# B&R Automation Studio project DivertAlignmentTool (part 3)

#### WriteDivertTransform.st - not listed in the package file held
```iecst
(*********************************************************************************
 * Copyright: B&R Industrial Automation GmbH
 * Author:    nealj
 * Created:   November 30, 2023/4:29 PM
 *
 *********************************************************************************)

FUNCTION WriteDivertTransform
	// Clear the transform
	brsmemset(ADR(Schematic.Svg.Transform),0,SIZEOF(Schematic.Svg.Transform));
	// Add the opening bracket
	Schematic.Svg.Transform := '[';
	// Find the first filled divert entry and set its color
	FOR i:=0 TO NUM_DIVERTS DO
		IF Schematic.Diverts[i].Overlap <> 0 THEN
			RectName.Value := i;
			RectName.String := INT_TO_STRING(RectName.Value);
			brsmemset(ADR(NewLine),0,SIZEOF(NewLine));
			NewLine := '{"select":"#Div_';
			NewLine := CONCAT(NewLine,RectName.String);
			// If not found yet, set grey (0)
			IF NOT Schematic.Diverts[i].Found THEN
				NewLine := CONCAT(NewLine,'","fill":0,"duration":0}');
			// If found, but not measured, set blue (1)
			ELSIF Schematic.Diverts[i].Found AND NOT Schematic.Diverts[i].Measurements.Measured THEN
				NewLine := CONCAT(NewLine,'","fill":1,"duration":0}');
			// If found and measured, set blue (1)
			ELSIF Schematic.Diverts[i].Found AND Schematic.Diverts[i].Measurements.Measured THEN
				NewLine := CONCAT(NewLine,'","fill":2,"duration":0}');
			END_IF
			brsstrcat(ADR(Schematic.Svg.Transform),ADR(NewLine));
			EXIT;
		END_IF
	END_FOR
	// For all subsequent diverts, set the color
	FOR i:=(i+1) TO NUM_DIVERTS DO
		IF Schematic.Diverts[i].Overlap <> 0 THEN
			RectName.Value := i;
			RectName.String := INT_TO_STRING(RectName.Value);
			brsmemset(ADR(NewLine),0,SIZEOF(NewLine));
			NewLine := ',{"select":"#Div_';					// <-- Note the comma at the front of the string to separate it from the previous transform
			NewLine := CONCAT(NewLine,RectName.String);
			// If not found yet, set grey (0)
			IF NOT Schematic.Diverts[i].Found THEN
				NewLine := CONCAT(NewLine,'","fill":0,"duration":0}');
				// If found, but not measured, set blue (1)
			ELSIF Schematic.Diverts[i].Found AND NOT Schematic.Diverts[i].Measurements.Measured THEN
				NewLine := CONCAT(NewLine,'","fill":1,"duration":0}');
				// If found and measured, set blue (1)
			ELSIF Schematic.Diverts[i].Found AND Schematic.Diverts[i].Measurements.Measured THEN
				NewLine := CONCAT(NewLine,'","fill":2,"duration":0}');
			END_IF
			brsstrcat(ADR(Schematic.Svg.Transform),ADR(NewLine));
		END_IF
	END_FOR
	// Add the closing bracket
	NewLine := ']';
	brsstrcat(ADR(Schematic.Svg.Transform),ADR(NewLine));

END_FUNCTION
```

### SampleTrakCode.var - Variables for the example trak program
```iecst
(*
Array of all segment references*)
VAR
	SegmentRefs : ARRAY[0..NUM_SEGMENTS] OF UDINT;
END_VAR
(*
Motion Parameters*)
VAR
	MotionParameters : ShMotionParType;
END_VAR
```

### Program Logical/SampleTrakCode/AssemblyCtrl (IEC) - The main task for the example trak program

#### Cyclic.st - Cyclic code
```iecst
PROGRAM _CYCLIC

	CASE AsmState OF

		// When the controller starts up, power on the trak
		ASM_IDLE:
			AsmReadInfo.Enable := TRUE;
			AsmReadStatus.Enable := TRUE;
			AsmState := ASM_POWER_ON;

		// If needed, power on the assembly and wait for it to power on
		ASM_POWER_ON:
			IF NOT AsmReadInfo.AssemblyInfo.PowerOn THEN
				AsmPowerOn.Execute := TRUE;
			ELSIF AsmReadInfo.AssemblyInfo.PowerOn AND AsmReadStatus.AssemblyReady THEN
				AsmPowerOn.Execute := FALSE;
				AsmState := ASM_FIND_ALL_SHUTTLES;
			END_IF

		// Wait for the start command, then get a list of all shuttles on the trak. Skip to ASM_RUNNING if there are no shuttles
		ASM_FIND_ALL_SHUTTLES:
			IF gStartTrak THEN
				AsmGetShuttle.Enable := TRUE;
				IF AsmGetShuttle.Valid THEN
					IF AsmGetShuttle.TotalCount > 0 THEN
						AsmState := ASM_READ_FROM_SHUTTLE;
					ELSE
						AsmGetShuttle.Enable := FALSE;
						AsmState := ASM_RUNNING;
					END_IF
				END_IF
			END_IF

		ASM_READ_FROM_SHUTTLE:
			AsmGetShuttle.Next := FALSE;
			// Read the userdata from the shuttle
			ShCopyUserData.Axis := ADR(AsmGetShuttle.Axis);
			ShCopyUserData.DataAddress := ADR(UserData);
			ShCopyUserData.DataSize := SIZEOF(UserData);
			ShCopyUserData.Mode := mcACPTRAK_USERDATA_GET;
			ShCopyUserData.Execute := TRUE;
			IF ShCopyUserData.Done THEN
				ShCopyUserData.Execute := FALSE;
				AsmState := ASM_WRITE_TO_SHUTTLE;
			END_IF

		// Make the shuttle grey, set its destination, and assign it a serial number
		ASM_WRITE_TO_SHUTTLE:
			// Set up intital userdata
			UserData.Red := 0.5;
			UserData.Green := 0.5;
			UserData.Blue := 0.5;
			IF UserData.ShuttleSerialNum = '' THEN
				SN_String := '';
				SN_Index := SN_Index + 1;
				SN_IndexStr := USINT_TO_STRING(SN_Index);
				SN_String := CONCAT(SN_String,SN_Prefix);
				SN_String := CONCAT(SN_String,SN_IndexStr);
				UserData.ShuttleSerialNum := SN_String;
			END_IF
			// Write the userdata to the shuttle
			ShCopyUserData.Axis := ADR(AsmGetShuttle.Axis);
			ShCopyUserData.DataAddress := ADR(UserData);
			ShCopyUserData.DataSize := SIZEOF(UserData);
			ShCopyUserData.Mode := mcACPTRAK_USERDATA_SET;
			ShCopyUserData.Execute := TRUE;
			IF ShCopyUserData.Done THEN
				ShCopyUserData.Execute := FALSE;
				AsmState := ASM_MOVE_SHUTTLE;
			END_IF

		// Send the shuttle to the destination defined above
		ASM_MOVE_SHUTTLE:
			RoutedMoveAbs.Axis := ADR(AsmGetShuttle.Axis);
			RoutedMoveAbs.Sector := ADR(SEC_MainLoop);
			RoutedMoveAbs.Position := 0.00;
			RoutedMoveAbs.Velocity := MotionParameters.Velocity;
			RoutedMoveAbs.Acceleration := MotionParameters.Acceleration;
			RoutedMoveAbs.Deceleration := MotionParameters.Deceleration;
			RoutedMoveAbs.AdvancedParameters.StartDirection := mcDIR_POSITIVE;
			RoutedMoveAbs.AdvancedParameters.EndDirection := mcDIR_POSITIVE;
			RoutedMoveAbs.AdvancedParameters.NumberOfTransitPoints := 0;
			RoutedMoveAbs.Execute := TRUE;
			AsmState := ASM_CHECK_FOR_MORE;

		// Once the move is active, check for remaining shuttles
		ASM_CHECK_FOR_MORE:
			IF RoutedMoveAbs.Active THEN
				RoutedMoveAbs.Execute := FALSE;
				IF AsmGetShuttle.RemainingCount > 0 THEN
					AsmGetShuttle.Next := TRUE;
					AsmState := ASM_READ_FROM_SHUTTLE;
				ELSE
					AsmGetShuttle.Enable := FALSE;
					AsmState := ASM_RUNNING;
				END_IF
			END_IF

		// All shuttles have been put in motion
		ASM_RUNNING:
			// Reset the start command
			gStartTrak := FALSE;
			// If the stop command is issued, stop all shuttles
			IF gStopTrak THEN
				AsmStop.Execute := TRUE;
				IF AsmStop.Done THEN
					AsmStop.Execute := FALSE;
					AsmState := ASMSTOP_FIND_ALL_SHUTTLES;
				END_IF
			END_IF

		// ===========================================================
		// GET ALL SHUTTLES TO BE STOPPED AT THE START OF THE TOP LOOP
		// ===========================================================
		// Get a list of all shuttles on the trak. Skip to ASM_RUNNING if there are no shuttles
		ASMSTOP_FIND_ALL_SHUTTLES:
			AsmGetShuttle.Enable := TRUE;
			IF AsmGetShuttle.Valid THEN
				IF AsmGetShuttle.TotalCount > 0 THEN
					AsmState := ASMSTOP_READ_FROM_SHUTTLE;
				ELSE
					AsmGetShuttle.Enable := FALSE;
					gStopTrak := FALSE;
					AsmState := ASM_IDLE;
				END_IF
			END_IF

		ASMSTOP_READ_FROM_SHUTTLE:
			AsmGetShuttle.Next := FALSE;
			// Read the userdata from the shuttle
			ShCopyUserData.Axis := ADR(AsmGetShuttle.Axis);
			ShCopyUserData.DataAddress := ADR(UserData);
			ShCopyUserData.DataSize := SIZEOF(UserData);
			ShCopyUserData.Mode := mcACPTRAK_USERDATA_GET;
			ShCopyUserData.Execute := TRUE;
			IF ShCopyUserData.Done THEN
				ShCopyUserData.Execute := FALSE;
				AsmState := ASMSTOP_WRITE_TO_SHUTTLE;
			END_IF

		// Make the shuttle black, and set its destination
		ASMSTOP_WRITE_TO_SHUTTLE:
			// Set userdata to reflect the stop
			UserData.Red := 0.0;
			UserData.Green := 0.0;
			UserData.Blue := 0.0;
			// Write the userdata to the shuttle
			ShCopyUserData.Axis := ADR(AsmGetShuttle.Axis);
			ShCopyUserData.DataAddress := ADR(UserData);
			ShCopyUserData.DataSize := SIZEOF(UserData);
			ShCopyUserData.Mode := mcACPTRAK_USERDATA_SET;
			ShCopyUserData.Execute := TRUE;
			IF ShCopyUserData.Done THEN
				ShCopyUserData.Execute := FALSE;
				AsmState := ASMSTOP_MOVE_SHUTTLE;
			END_IF

		// Send the shuttle to the destination defined above
		ASMSTOP_MOVE_SHUTTLE:
			RoutedMoveAbs.Axis := ADR(AsmGetShuttle.Axis);
			RoutedMoveAbs.Sector := ADR(SEC_MainLoop);
			RoutedMoveAbs.Position := 0.00;
			RoutedMoveAbs.Velocity := MotionParameters.Velocity;
			RoutedMoveAbs.Acceleration := MotionParameters.Acceleration;
			RoutedMoveAbs.Deceleration := MotionParameters.Deceleration;
			RoutedMoveAbs.AdvancedParameters.StartDirection := mcDIR_UNDEFINED;
			RoutedMoveAbs.AdvancedParameters.EndDirection := mcDIR_POSITIVE;
			RoutedMoveAbs.Execute := TRUE;
			AsmState := ASMSTOP_CHECK_FOR_MORE;

		// Once the move is active, check for remaining shuttles
		ASMSTOP_CHECK_FOR_MORE:
			IF RoutedMoveAbs.Active THEN
				RoutedMoveAbs.Execute := FALSE;
				IF AsmGetShuttle.RemainingCount > 0 THEN
					AsmGetShuttle.Next := TRUE;
					AsmState := ASMSTOP_READ_FROM_SHUTTLE;
				ELSE
					AsmGetShuttle.Enable := FALSE;
					gStopTrak := FALSE;
					AsmState := ASM_IDLE;
				END_IF
			END_IF

		// Example error state
		ASM_ERROR:

	END_CASE

	// Call FUBs
	AsmPowerOn();
	AsmPowerOff();
	AsmReadInfo();
	AsmReadStatus();
	AsmGetShuttle();
	AsmStop();
	ShCopyUserData();
	RoutedMoveAbs();
	SecAddShuttle();

END_PROGRAM
```

#### Init.st - Init code
```iecst
PROGRAM _INIT

	// Set up assembly FUBs
	AsmPowerOn.Assembly := ADR(gAssembly_1);
	AsmPowerOff.Assembly := ADR(gAssembly_1);
	AsmReadInfo.Assembly := ADR(gAssembly_1);
	AsmReadStatus.Assembly := ADR(gAssembly_1);
	AsmGetShuttle.Assembly := ADR(gAssembly_1);
	AsmStop.Assembly := ADR(gAssembly_1);
	AsmStop.StopMode := mcSTOPMODE_JERK_LIMIT;

	//Set up shuttle spawning FUB
	SecAddShuttle.Sector := ADR(SEC_MainLoop);
	SecAddShuttle.Position := 0.00;

	// Set motion parameters
	MotionParameters.Velocity     := 1.0;
	MotionParameters.Acceleration := 40.0;
	MotionParameters.Deceleration := 40.0;

	// List all segment references
	SegmentRefs[1] := ADR(SEG_001);
	SegmentRefs[2] := ADR(SEG_002);
	SegmentRefs[3] := ADR(SEG_003);
	SegmentRefs[4] := ADR(SEG_004);
	SegmentRefs[5] := ADR(SEG_005);
	SegmentRefs[6] := ADR(SEG_006);
	SegmentRefs[7] := ADR(SEG_007);
	SegmentRefs[8] := ADR(SEG_008);
	SegmentRefs[9] := ADR(SEG_009);
	SegmentRefs[10] := ADR(SEG_010);
	SegmentRefs[11] := ADR(SEG_011);
	SegmentRefs[12] := ADR(SEG_012);
	SegmentRefs[13] := ADR(SEG_013);
	SegmentRefs[14] := ADR(SEG_014);
	SegmentRefs[15] := ADR(SEG_015);
	SegmentRefs[16] := ADR(SEG_016);
	SegmentRefs[17] := ADR(SEG_017);
	SegmentRefs[18] := ADR(SEG_018);
	SegmentRefs[19] := ADR(SEG_019);
	SegmentRefs[20] := ADR(SEG_020);
	SegmentRefs[21] := ADR(SEG_021);
	SegmentRefs[22] := ADR(SEG_022);
	SegmentRefs[23] := ADR(SEG_023);
	SegmentRefs[24] := ADR(SEG_024);
	SegmentRefs[25] := ADR(SEG_025);
	SegmentRefs[26] := ADR(SEG_026);
	SegmentRefs[27] := ADR(SEG_027);
	SegmentRefs[28] := ADR(SEG_028);
	SegmentRefs[29] := ADR(SEG_029);
	SegmentRefs[30] := ADR(SEG_030);
	SegmentRefs[31] := ADR(SEG_031);
	SegmentRefs[32] := ADR(SEG_032);
	SegmentRefs[33] := ADR(SEG_033);
	SegmentRefs[34] := ADR(SEG_034);
	SegmentRefs[35] := ADR(SEG_035);
	SegmentRefs[36] := ADR(SEG_036);
	SegmentRefs[37] := ADR(SEG_037);
	SegmentRefs[38] := ADR(SEG_038);
	SegmentRefs[39] := ADR(SEG_039);
	SegmentRefs[40] := ADR(SEG_040);
	SegmentRefs[41] := ADR(SEG_041);
	SegmentRefs[42] := ADR(SEG_042);
	SegmentRefs[43] := ADR(SEG_043);
	SegmentRefs[44] := ADR(SEG_044);
	SegmentRefs[45] := ADR(SEG_045);
	SegmentRefs[46] := ADR(SEG_046);
	SegmentRefs[47] := ADR(SEG_047);
	SegmentRefs[48] := ADR(SEG_048);
	SegmentRefs[49] := ADR(SEG_049);
	SegmentRefs[50] := ADR(SEG_050);
	SegmentRefs[51] := ADR(SEG_051);
	SegmentRefs[52] := ADR(SEG_052);
	SegmentRefs[53] := ADR(SEG_053);
	SegmentRefs[54] := ADR(SEG_054);
	SegmentRefs[55] := ADR(SEG_055);
	SegmentRefs[56] := ADR(SEG_056);
	SegmentRefs[57] := ADR(SEG_057);
	SegmentRefs[58] := ADR(SEG_058);
	SegmentRefs[59] := ADR(SEG_059);
	SegmentRefs[60] := ADR(SEG_060);
	SegmentRefs[61] := ADR(SEG_061);
	SegmentRefs[62] := ADR(SEG_062);
	SegmentRefs[63] := ADR(SEG_063);
	SegmentRefs[64] := ADR(SEG_064);
	SegmentRefs[65] := ADR(SEG_065);
	SegmentRefs[66] := ADR(SEG_066);
	SegmentRefs[67] := ADR(SEG_067);
	SegmentRefs[68] := ADR(SEG_068);
	SegmentRefs[69] := ADR(SEG_069);
	SegmentRefs[70] := ADR(SEG_070);
	SegmentRefs[71] := ADR(SEG_071);
	SegmentRefs[72] := ADR(SEG_072);
	SegmentRefs[73] := ADR(SEG_073);
	SegmentRefs[74] := ADR(SEG_074);
	SegmentRefs[75] := ADR(SEG_075);
	SegmentRefs[76] := ADR(SEG_076);
	SegmentRefs[77] := ADR(SEG_077);
	SegmentRefs[78] := ADR(SEG_078);
	SegmentRefs[79] := ADR(SEG_079);
	SegmentRefs[80] := ADR(SEG_080);
	SegmentRefs[81] := ADR(SEG_081);
	SegmentRefs[82] := ADR(SEG_082);
	SegmentRefs[83] := ADR(SEG_083);

	// List of all sectors (to avoid warnings in the logger)
	SEC_MainLoop;
	SEC_RedHerring_1;
	SEC_SecondLoop;
	SEC_VolcanoLeft;
	SEC_VolcanoRight;
	SEC_Squiggle;
	SEC_FlipFlop;
	SEC_RedHerring_2;
	SEC_MaintenanceLoop;

END_PROGRAM
```

#### Types.typ - Local data types
```iecst
TYPE
	AsmStateEnum :
		( (*State of the assembly control task*)
		ASM_IDLE,
		ASM_POWER_ON,
		ASM_FIND_ALL_SHUTTLES,
		ASM_READ_FROM_SHUTTLE,
		ASM_TRACK_SHUTTLE,
		ASM_WRITE_TO_SHUTTLE,
		ASM_MOVE_SHUTTLE,
		ASM_CHECK_FOR_MORE,
		ASM_RUNNING,
		ASMSTOP_FIND_ALL_SHUTTLES,
		ASMSTOP_READ_FROM_SHUTTLE,
		ASMSTOP_WRITE_TO_SHUTTLE,
		ASMSTOP_MOVE_SHUTTLE,
		ASMSTOP_CHECK_FOR_MORE,
		ASM_ERROR
		);
END_TYPE
```

#### Variables.var - Local variables
```iecst
(*Assembly variables*)
VAR
	AsmPowerOn : MC_BR_AsmPowerOn_AcpTrak; (*FUB to power on the assembly*)
	AsmPowerOff : MC_BR_AsmPowerOff_AcpTrak; (*FUB to power off the assembly*)
	AsmReadInfo : MC_BR_AsmReadInfo_AcpTrak; (*FUB to read the information of the assembly*)
	AsmReadStatus : MC_BR_AsmReadStatus_AcpTrak; (*FUB to read the status of the assembly*)
	AsmGetShuttle : MC_BR_AsmGetShuttle_AcpTrak; (*FUB to get references for all shuttles on the assembly*)
	AsmStop : MC_BR_AsmStop_AcpTrak; (*FUB to get references for all shuttles on the assembly*)
	AsmState : AsmStateEnum; (*State of the assembly control task*)
	SecAddShuttle : MC_BR_SecAddShuttle_AcpTrak;
END_VAR
(*
Shuttle variables*)
VAR
	ShCopyUserData : MC_BR_ShCopyUserData_AcpTrak; (*FUB for the initial writing of data during startup*)
	UserData : UserDataType; (*Structure for the initial writing of data during startup*)
	RoutedMoveAbs : MC_BR_RoutedMoveAbs_AcpTrak; (*FUB to move the shuttles on the trak to their first station*)
END_VAR
(*
Variables for serial number generation*)
VAR
	SN_Prefix : STRING[9] := 'TEST_SN_'; (*The prefix for all generated serial numbers*)
	SN_Index : USINT := 0; (*The number to be assigned to each shuttle (as a number)*)
	SN_IndexStr : STRING[4]; (*The number to be assigned to each shuttle (as a string)*)
	SN_String : STRING[12]; (*The string of the serial number to be assigned to each shuttle*)
END_VAR
```

#### Exit.st
```iecst
PROGRAM _EXIT

	RoutedMoveAbs.Execute := FALSE;
	RoutedMoveAbs();

END_PROGRAM
```

### Program Logical/DivertAlignment/GatherInfo (IEC)

#### Types.typ
```iecst
TYPE
	GatherStateEnum :
		(
		GATHER_IDLE,
		GATHER_SEG_AND_SEC,
		GATHER_SEG_AND_SEC_INFO,
		GATHER_DIVERTS,
		GATHER_SHUTTLE,
		GATHER_MOVE_TO_START,
		GATHER_MOVE_ALONG_SEC,
		GATHER_MONITOR_FOR_MIDPOINT,
		GATHER_ACKNOWLEDGE,
		GATHER_DONE
		);
END_TYPE
```

#### Variables.var
```iecst
VAR
	GatherState : GatherStateEnum;
	AssemblySchematics : AsmSchemType;
END_VAR
(*
FUBs and Vars for getting segments and their information*)
VAR
	AsmGetSeg : MC_BR_AsmGetSegment_AcpTrak;
	SecStop : MC_BR_SecStop_AcpTrak;
	SegGetInfo : MC_BR_SegGetInfo_AcpTrak;
	SecGetInfo : MC_BR_SecGetInfo_AcpTrak;
	CmdGather : BOOL;
	CmdContinue : BOOL;
	AsmGetSec : MC_BR_AsmGetSector_AcpTrak;
END_VAR
(*
FUBs and Vars for moving the shuttle around the trak*)
VAR
	AsmGetShuttle : MC_BR_AsmGetShuttle_AcpTrak;
	RoutedMoveAbs : MC_BR_RoutedMoveAbs_AcpTrak;
	ElasticMoveAbs : MC_BR_ElasticMoveAbs_AcpTrak;
	ShReadInfo : MC_BR_ShReadInfo_AcpTrak;
	ShReadSeg : MC_BR_ShReadSegmentInfo_AcpTrak;
	TestVelocity : REAL := 1.0;
	DivertIndex : UINT;
	SectorIndex : UINT;
	AcknowledgeTimer : TON;
	AcknowledgeTime : TIME := T#400ms;
END_VAR
```

#### Cyclic.st
```iecst
PROGRAM _CYCLIC
	(* Insert code here *)
	CASE GatherState OF
		GATHER_IDLE:
			// Wait for command, then clear the schematic structure and enable the AsmGetSeg and AsmGetSec FUBs
			IF CmdGather THEN
				brsmemset(ADR(AssemblySchematics),0,SIZEOF(AssemblySchematics));
				AsmGetSeg.Enable := TRUE;
				AsmGetSec.Enable := TRUE;
				GatherState := GATHER_SEG_AND_SEC;
			END_IF

		GATHER_SEG_AND_SEC:
			// Wait for validity
			IF AsmGetSeg.Valid AND AsmGetSec.Valid THEN
				// Clear the "next" signals
				AsmGetSeg.Next := FALSE;
				AsmGetSec.Next := FALSE;
				// Plug the segment and sectors into the respective get infor FUBs
				SegGetInfo.Segment := ADR(AsmGetSeg.Segment);
				SecGetInfo.Sector := ADR(AsmGetSec.Sector);
				// Execute the FUBs
				SegGetInfo.Execute := TRUE;
				SecGetInfo.Execute := TRUE;
				GatherState := GATHER_SEG_AND_SEC_INFO;
			END_IF

		GATHER_SEG_AND_SEC_INFO:
			// Wait for the SegGetInfo and SecGetInfo FUBs to finish
			IF SegGetInfo.Done AND SecGetInfo.Done THEN
				// Record the segment information (use the segment ID as the index)
				AssemblySchematics.Segment[SegGetInfo.SegmentInfo.ID].Reference := AsmGetSeg.Segment;
				AssemblySchematics.Segment[SegGetInfo.SegmentInfo.ID].Name := SegGetInfo.SegmentInfo.Name;
				AssemblySchematics.Segment[SegGetInfo.SegmentInfo.ID].ID := SegGetInfo.SegmentInfo.ID;
				AssemblySchematics.Segment[SegGetInfo.SegmentInfo.ID].Type := SegGetInfo.SegmentInfo.Type;
				AssemblySchematics.Segment[SegGetInfo.SegmentInfo.ID].StartFrame := SegGetInfo.SegmentInfo.StartFrame;
				AssemblySchematics.Segment[SegGetInfo.SegmentInfo.ID].EndFrame := SegGetInfo.SegmentInfo.EndFrame;
				// Record the sector information (store them in the order they are found)
				AssemblySchematics.Sectors[AsmGetSec.TotalCount - AsmGetSec.RemainingCount - 1].Reference := AsmGetSec.Sector;
				AssemblySchematics.Sectors[AsmGetSec.TotalCount - AsmGetSec.RemainingCount - 1].Name := SecGetInfo.SectorInfo.Name;
				AssemblySchematics.Sectors[AsmGetSec.TotalCount - AsmGetSec.RemainingCount - 1].Length := SecGetInfo.SectorInfo.Length;
				AssemblySchematics.Sectors[AsmGetSec.TotalCount - AsmGetSec.RemainingCount - 1].Type := SecGetInfo.SectorInfo.Type;
				// Reset the execute commands
				SegGetInfo.Execute := FALSE;
				SecGetInfo.Execute := FALSE;
				// If there are more segments, iterate
				IF AsmGetSeg.RemainingCount > 0 THEN
					AsmGetSeg.Next := TRUE;
					GatherState := GATHER_SEG_AND_SEC;
				END_IF
				// If there are more sectors, iterate
				IF AsmGetSec.RemainingCount > 0 THEN
					AsmGetSec.Next := TRUE;
					GatherState := GATHER_SEG_AND_SEC;
				END_IF
				// If there are no more segments and no more sectors, the task is done
				IF AsmGetSeg.RemainingCount = 0 AND AsmGetSec.RemainingCount = 0 THEN
					AsmGetSeg.Enable := FALSE;
					AsmGetSec.Enable := FALSE;
					GatherState := GATHER_DIVERTS;
				END_IF
			END_IF

		GATHER_DIVERTS:
			// Use the CheckForDiverts function
			CheckForDiverts(ADR(AssemblySchematics));
			GatherState := GATHER_SHUTTLE;

		GATHER_SHUTTLE:
			// Get the reference of the shuttle on the trak
			AsmGetShuttle.Enable := TRUE;
			IF AsmGetShuttle.Valid THEN
				RoutedMoveAbs.Axis := ADR(AsmGetShuttle.Axis);
				ShReadInfo.Axis := ADR(AsmGetShuttle.Axis);
				ShReadInfo.Enable := TRUE;
				ShReadSeg.Axis := ADR(AsmGetShuttle.Axis);
				ShReadSeg.Enable := TRUE;
				GatherState := GATHER_MOVE_TO_START;
			END_IF

		GATHER_MOVE_TO_START:
			// ! ! ! ! ! ! ! ! ! ! ! ! ! ! ! ! ! ! ! ! ! ! ! ! ! ! ! ! ! ! ! ! ! ! ! ! ! !
			// ! ! ! ! ! ! ! ! ! ! ! ! ! ! ! ! ! ! ! ! ! ! ! ! ! ! ! ! ! ! ! ! ! ! ! ! ! !
			// ! ! !  CHANGE THE STATES SO THAT DIVERTS CAN BE FOUND ON ROUTES TOO   ! ! !
			// ! ! ! ! ! ! ! ! ! ! ! ! ! ! ! ! ! ! ! ! ! ! ! ! ! ! ! ! ! ! ! ! ! ! ! ! ! !
			// ! ! !           MAKE SHUTTLE CHANGE COLOR WHEN DIVERT FOUND           ! ! !
			// ! ! ! ! ! ! ! ! ! ! ! ! ! ! ! ! ! ! ! ! ! ! ! ! ! ! ! ! ! ! ! ! ! ! ! ! ! !
			// ! ! ! ! ! ! ! ! ! ! ! ! ! ! ! ! ! ! ! ! ! ! ! ! ! ! ! ! ! ! ! ! ! ! ! ! ! !

			// Move to the start of the sector at full speed
			RoutedMoveAbs.Sector := ADR(AssemblySchematics.Sectors[SectorIndex].Reference);
			RoutedMoveAbs.Axis := ADR(AsmGetShuttle.Axis);
			RoutedMoveAbs.Position := 0;
			RoutedMoveAbs.Velocity := 4;
			RoutedMoveAbs.Acceleration := 40;
			RoutedMoveAbs.Deceleration := 40;
			RoutedMoveAbs.AdvancedParameters.StartDirection := mcDIR_UNDEFINED;
			RoutedMoveAbs.AdvancedParameters.EndDirection := mcDIR_UNDEFINED;
			RoutedMoveAbs.AdvancedParameters.ShuttleOrientation := mcDIR_UNDEFINED;
			RoutedMoveAbs.Execute := TRUE;
			IF RoutedMoveAbs.Done THEN
				RoutedMoveAbs.Execute := FALSE;
				GatherState := GATHER_MOVE_ALONG_SEC;
			END_IF

		GATHER_MOVE_ALONG_SEC:
			// Move to the end of the sector in the positive direction
			ElasticMoveAbs.Axis := ADR(AsmGetShuttle.Axis);
			ElasticMoveAbs.Position := AssemblySchematics.Sectors[SectorIndex].Length;
			ElasticMoveAbs.Velocity := TestVelocity;
			ElasticMoveAbs.Acceleration := 40;
			ElasticMoveAbs.Deceleration := 40;
			ElasticMoveAbs.Execute := TRUE;
			IF ElasticMoveAbs.Active THEN
				GatherState := GATHER_MONITOR_FOR_MIDPOINT;
			END_IF

		GATHER_MONITOR_FOR_MIDPOINT:
			// Constantly compare the current seg position to the divert seg midpoints
			// Execute a stop if within DIV_MIDPOINT_TOLERANCE of one
			FOR DivertIndex:=0 TO NUM_DIVERTS DO
				IF NOT AssemblySchematics.Diverts[DivertIndex].Measured THEN
					// If the shuttle is on the same segment as the divert's first segment then compare the positions
					IF (ShReadInfo.ShuttleInfo.CurrentValues.SegmentPosition.Name = AssemblySchematics.Diverts[DivertIndex].SegName[0]) THEN
						// If the shuttles current position on the segment is within DIV_MIDPOINT_TOLERANCE of the midpoint then stop and take the measurement
						IF (ShReadInfo.ShuttleInfo.CurrentValues.SegmentPosition.Position > AssemblySchematics.Diverts[DivertIndex].DivertMid[0] - DIV_MIDPOINT_TOLERANCE) AND
							(ShReadInfo.ShuttleInfo.CurrentValues.SegmentPosition.Position < AssemblySchematics.Diverts[DivertIndex].DivertMid[0] + DIV_MIDPOINT_TOLERANCE) THEN
							AssemblySchematics.Diverts[DivertIndex].Measured := TRUE;
							ElasticMoveAbs.Execute := FALSE;
							SecStop.Sector := ADR(AssemblySchematics.Sectors[SectorIndex].Reference);
							SecStop.Execute := TRUE;
							GatherState := GATHER_ACKNOWLEDGE;
							EXIT;
						END_IF
					// If the shuttle is on the same segment as the divert's second segment then compare the positions
					ELSIF (ShReadInfo.ShuttleInfo.CurrentValues.SegmentPosition.Name = AssemblySchematics.Diverts[DivertIndex].SegName[1]) THEN
						// If the shuttles current position on the segment is within DIV_MIDPOINT_TOLERANCE of the midpoint then stop and take the measurement
						IF (ShReadInfo.ShuttleInfo.CurrentValues.SegmentPosition.Position > AssemblySchematics.Diverts[DivertIndex].DivertMid[1] - DIV_MIDPOINT_TOLERANCE) AND
							(ShReadInfo.ShuttleInfo.CurrentValues.SegmentPosition.Position < AssemblySchematics.Diverts[DivertIndex].DivertMid[1] + DIV_MIDPOINT_TOLERANCE) THEN
							AssemblySchematics.Diverts[DivertIndex].Measured := TRUE;
							ElasticMoveAbs.Execute := FALSE;
							SecStop.Sector := ADR(AssemblySchematics.Sectors[SectorIndex].Reference);
							SecStop.Execute := TRUE;
							GatherState := GATHER_ACKNOWLEDGE;
							EXIT;
						END_IF
					END_IF
				END_IF
			END_FOR
			// If the move finishes, the shuttle reached the end of the sector. Increment the sector index
			IF ElasticMoveAbs.Done THEN
				ElasticMoveAbs.Execute := FALSE;
				SectorIndex := SectorIndex + 1;
				// if the index is less than or equal to the limit, check that it is not an empty entry
				IF SectorIndex <= NUM_SECTORS THEN
					// If the entry is not empty, go to the start of that sector
					IF AssemblySchematics.Sectors[SectorIndex].Length <> 0 THEN
						GatherState := GATHER_MOVE_TO_START;
					// If the entry is empty, all sectors have been checked
					ELSE
						GatherState := GATHER_DONE;
					END_IF
				// If the index is greater than the limit, all entries have been checked
				ELSE
					GatherState := GATHER_DONE;
				END_IF
			END_IF

		GATHER_ACKNOWLEDGE:
			// When the command is given, go back to moving along the sector
			IF SecStop.Done THEN
				SecStop.Execute := FALSE;
				AcknowledgeTimer.PT := AcknowledgeTime;
				AcknowledgeTimer.IN := TRUE;
			END_IF
			IF AcknowledgeTimer.Q THEN
				AcknowledgeTimer.IN := FALSE;
				GatherState := GATHER_MOVE_ALONG_SEC;
			END_IF

		GATHER_DONE:
			DivertIndex := 0;
			SectorIndex := 0;
			IF NOT CmdGather THEN
				GatherState := GATHER_IDLE;
			END_IF

	END_CASE

	AsmGetSeg();
	AsmGetSec();
	SecStop();
	SegGetInfo();
	SecGetInfo();
	AsmGetShuttle();
	RoutedMoveAbs();
	ElasticMoveAbs();
	ShReadInfo();
	ShReadSeg();
	AcknowledgeTimer();

END_PROGRAM
```

#### Init.st
```iecst
PROGRAM _INIT

	AsmGetSeg.Assembly := ADR(gAssembly_1);
	AsmGetSec.Assembly := ADR(gAssembly_1);
	AsmGetShuttle.Assembly := ADR(gAssembly_1);

END_PROGRAM
```

- Visualisation Logical/mappView (not shown)

Listed in the project but not available here: Logical/Global.typ, Logical/Libraries/TrkBufLib/Types.typ, Logical/Libraries/TrkBufLib/Constants.var, Logical/Libraries/TrkBufLib/TrkBufLib.fun, Logical/Libraries/TrkBufLib/RoutedMoveVelTrigBuffer.st, Logical/Libraries/TrkBufLib/ElasticMoveAbsPosBuffer.st, Logical/Libraries/TrkBufLib/BufferAddSh.st, Logical/Libraries/TrkBufLib/BufferGetFirst.st, Logical/Libraries/TrkBufLib/BufferRemoveFirst.st, Logical/Libraries/TrkBufLib/ShInBuffer.st, Logical/Libraries/TrkBufLib/BufferShAvailable.st, Logical/SampleTrakCode/SampleTrakCode.typ
